FUNCTION_BLOCK FB_DynamicFifo
VAR
	/// Configuration
	_bFreeDataPointer		: BOOL;
	/// Actual Count of the elements in the buffer
	_uinItemCount			: UINT;
	/// Index of the first added element
	_pFirstElement			: POINTER TO T_QueueBase;
	/// Index of the last added element
	_pLastElement			: POINTER TO T_QueueBase;
	/// Limit the queue size  0=NO-LIMIT
	_uinQueueLimit			: UINT := 0;
	/// Behavior when the queue is full FALSE=Do not add any item if full, TRUE= Delete the oldest one and add the new one.
	_bolRingBuffer			: BOOL := FALSE;
END_VAR

{attribute 'object_name' := 'Pop'}
METHOD Pop : POINTER TO BYTE
VAR
	pItem: POINTER TO T_QueueBase;
END_VAR
Pop := TC3_MEMMAN.NULL;

IF _uinItemCount > 0 THEN
	pItem := _pFirstElement;
	
	_pFirstElement := _pFirstElement^.pNext;

	IF _pFirstElement <> TC3_MEMMAN.NULL THEN
		_pFirstElement^.pPrevious := TC3_MEMMAN.NULL;
	ELSE
		_pLastElement := TC3_MEMMAN.NULL;
	END_IF

	_uinItemCount := _uinItemCount - 1;

	Pop := pItem^.pData;
	__DELETE(pItem);
END_IF
END_METHOD

{attribute 'object_name' := 'Push'}
METHOD Push : INT
VAR_INPUT
	pData: POINTER TO BYTE;
END_VAR
VAR
	pItem: POINTER TO T_QueueBase;
END_VAR
IF (_uinQueueLimit = 0) OR (_uinItemCount < _uinQueueLimit) OR ((_uinItemCount = _uinQueueLimit) AND _bolRingBuffer) THEN
	IF (_uinItemCount = _uinQueueLimit) AND _bolRingBuffer THEN
		Pop();
	END_IF	

	AddItem(pData);
	
	Push := UINT_TO_INT(_uinItemCount);
ELSE
	Push := -1;
END_IF
END_METHOD

METHOD PROTECTED AddItem : BOOL
VAR_INPUT
	pData: POINTER TO BYTE;
END_VAR
VAR
	pItem: POINTER TO T_QueueBase;
END_VAR
pItem := __NEW(T_QueueBase);
pItem^.pData := pData;

IF _uinItemCount = 0 THEN
	_pFirstElement := pItem;
	_pLastElement  := pItem;
	pItem^.pNext := TC3_MEMMAN.NULL;
	pItem^.pPrevious := TC3_MEMMAN.NULL;
ELSE
	_pLastElement^.pNext:= pItem;
	pItem^.pPrevious := _pLastElement;
	pItem^.pNext := TC3_MEMMAN.NULL;
	_pLastElement  := pItem;
END_IF

_uinItemCount := _uinItemCount + 1;
END_METHOD

PROPERTY PUBLIC RingBuffer : BOOL
SET
_bolRingBuffer := RingBuffer;
END_SET
GET
RingBuffer := _bolRingBuffer;
END_GET
END_PROPERTY

{attribute 'object_name' := 'Peek'}
METHOD Peek : POINTER TO BYTE
Peek := TC3_MEMMAN.NULL;

IF _uinItemCount > 0 THEN
	Peek := _pFirstElement^.pData;
END_IF
END_METHOD

PROPERTY PUBLIC QueueLimit : UINT
GET
QueueLimit := _uinQueueLimit;
END_GET
SET
_uinQueueLimit := QueueLimit;
END_SET
END_PROPERTY

PROPERTY FreeDataPointer : BOOL
SET
_bFreeDataPointer := FreeDataPointer;
END_SET
GET
FreeDataPointer := _bFreeDataPointer;
END_GET
END_PROPERTY

{attribute 'object_name' := 'ClearFifo'}
METHOD ClearFifo : BOOL
VAR
	pItem: POINTER TO T_QueueBase;
	pNextItem: POINTER TO T_QueueBase;
END_VAR
pItem := _pFirstElement;
_pFirstElement := NULL;

WHILE pItem <> TC3_MEMMAN.NULL DO
	pNextItem := pItem^.pNext;
	
	IF _bFreeDataPointer THEN
		__DELETE(pItem^.pData);
	END_IF
	
	__DELETE(pItem);
	pItem := pNextItem;
END_WHILE

_pLastElement := NULL;
_uinItemCount := 0;
END_METHOD

PROPERTY ItemCount : UINT
GET
ItemCount := _uinItemCount;
END_GET
END_PROPERTY

END_FUNCTION_BLOCK

(* stored: Version 1.1.0.1, ProductVersion 3.1.0.36
   POU FB_DynamicFifo: Id {775546da-d62a-4095-8834-9f828c0de9e5}, SpecialFunc None
   Method Pop: Id {24f665ed-39ef-4d05-a514-5b6e703f4f04}
   Method Push: Id {4ba242b0-7aec-4445-afd7-55552d74cb37}
   Method AddItem: Id {529ad006-3ac5-4bbe-bdc7-de0c2849ba14}
   Property RingBuffer: Id {73ecdfe2-b156-4280-8a87-46c390548293}
   Set Set: Id {295596ed-8e6f-47cd-a98e-73bdfb343ae4}
   Get Get: Id {ee21db1f-dbf3-4c26-b36d-b04ef9c87e3d}
   Method Peek: Id {855cb792-2fef-4a6a-97bb-b0c19f8c9d0b}
   Property QueueLimit: Id {d3167dbc-b3fb-4bb1-8b60-b962656f7676}
   Get Get: Id {0b11d454-da29-40b5-9b9c-bd4194a4579d}
   Set Set: Id {2352dc0c-296a-474f-871e-71385bfca5ed}
   Property FreeDataPointer: Id {d8615c9c-cc4e-4f68-8683-8ec365a63b21}
   Set Set: Id {ea585a2d-3864-4fdf-a45a-885e837a622b}
   Get Get: Id {ee2e23ab-c3ed-494b-8059-3ca4a2b48bcf}
   Method ClearFifo: Id {de691d59-86b0-441f-ac72-0cd22129d7cb}
   Property ItemCount: Id {fddbec3a-ffce-4ec3-b578-25480543f3b1}
   Get Get: Id {8e08995b-a44b-4e75-94a2-9ed99ad89545} *)
